Staubli VAL3: ISO_PDU_DATA_T.dtx

public num TPKT[4]
public num COPT[3]
public S7telegram_T S7telegram
  [0]
    num H[18]
    num DATA[240]
